{attribute addProperty BoxType "EL1918-0000-0016"}
{attribute addProperty Id "FSOEAT %Q*FSOE_F2812FEE486"}
{attribute addProperty CRC "1855391509"}
{attribute addProperty SizeInBites "48"}
{attribute addProperty SizeInBytes "6"}
TYPE FSoE_Outputs_6E970715 :
STRUCT
	{attribute addProperty Name "FSOE"}
	FSOE AT %Q* : FSOE_F2812FEE;
END_STRUCT
END_TYPE

(* stored: Version 1.2.0.0, ProductVersion 3.1.4024.9
   DUT FSoE_Outputs_6E970715: Id {07e7b112-af0f-4ecb-ba85-e4ca4f40f1b5} *)
